FUNCTION_BLOCK FB_PLCState
VAR_OUTPUT
	EL9410					AT %I* : ST_EL9410;
	get							: ST_PLCstate_get;
END_VAR
VAR
	ton_refreshpulse					: TON := (PT := T#500ms);
	events : ST_PLC_events;
	by_PNErrorsAllowed					: BYTE;
	ui_EthercatMasterState		AT %I* : UINT;
	ui_ProfinetNoErrorDevices	AT %I* : UINT;
	ui_ProfinetNoDiagDevices	AT %I* : UINT;
	ui_SafetyLogicState			AT %I* : UINT;	
	
	ton_SystemReady					: TON := (IN := FALSE, PT := T#15S);	
	
	fb_cpuload 						: TC_CpuUsage;
	
END_VAR

events.b_EthercatMasterFault := ui_EthercatMasterState <> 0;

ton_SystemReady(IN:= TRUE);
GVL.b_SystemReady	:= ton_SystemReady.Q;

IF settings.Configuration.e_PNcouplerType = 0 THEN
	by_PNErrorsAllowed := 3;
ELSE 
	by_PNErrorsAllowed := 2;
END_IF

// get cpu load
ton_refreshpulse(IN := NOT ton_refreshpulse.Q);
fb_cpuload(start:= ton_refreshpulse.Q,
	TMOUT:= T#5S);
get.r_CPUload:= TO_REAL(fb_cpuload.USAGE);

IF ui_ProfinetNoErrorDevices > by_PNErrorsAllowed THEN
	get.e_ProfinetState := eNetcomState.Error;
ELSIF ui_ProfinetNoDiagDevices > by_PNErrorsAllowed THEN
	get.e_ProfinetState := eNetcomState.Warning;
ELSIF ui_ProfinetNoErrorDevices <= by_PNErrorsAllowed AND ui_ProfinetNoDiagDevices <= by_PNErrorsAllowed THEN
	get.e_ProfinetState := eNetcomState.OK;
ELSE
	get.e_ProfinetState := eNetcomState.NotConnected;
END_IF

IF ui_EthercatMasterState = 0 THEN
	get.e_EthercatState := eNetcomState.OK;
ELSIF ui_EthercatMasterState = 1 THEN
	get.e_EthercatState := eNetcomState.NotConnected;
ELSE
	get.e_EthercatState := eNetcomState.Error;
END_IF

METHOD GetDiagnostics
VAR_IN_OUT
	AddError		: ARRAY [*] OF FB_AddErrorST;
	a_ActiveEvents	: ARRAY [*] OF ST_ErrorStruct;
	w_Index			: WORD;
END_VAR
(*PLC io supply fault*)		AddError[w_Index](
					b_ErrorTrig			:= EL9410.bit_UpUndervoltage OR EL9410.bit_UsUndervoltage,
					out_ST_Error			:= a_ActiveEvents[w_Index],
					w_ErrorID					:= 1,
					e_ObjectID				:= eObject_ID.PLC,
					s_Message				:= 'EL9410 supply fault',
					e_sev					:= eSeverity.Quickshutdown
				);
				w_Index := w_Index +1;
				
(*Ethercat master fault*)		AddError[w_Index](
					b_ErrorTrig			:= events.b_EthercatMasterFault,
					out_ST_Error			:= a_ActiveEvents[w_Index],
					w_ErrorID					:= 2,
					s_Message				:= 'Ethercat master fault',
					e_sev					:= eSeverity.normalshutdown,
				);
				w_Index := w_Index +1;
END_METHOD

END_FUNCTION_BLOCK

(* stored: Version 1.1.0.1, ProductVersion 3.1.4026.18
   POU FB_PLCState: Id {a13546c6-375c-4536-80f7-17a8eb8dfe7c}, SpecialFunc None
   Method GetDiagnostics: Id {696ad14c-cd40-409d-abeb-19d3ba8eea88} *)
